// Mitsubishi GX Works2 project: 시퀀스 부분 반복 회로 (카운터)   PLC: Q03UDV

PROGRAM MAIN
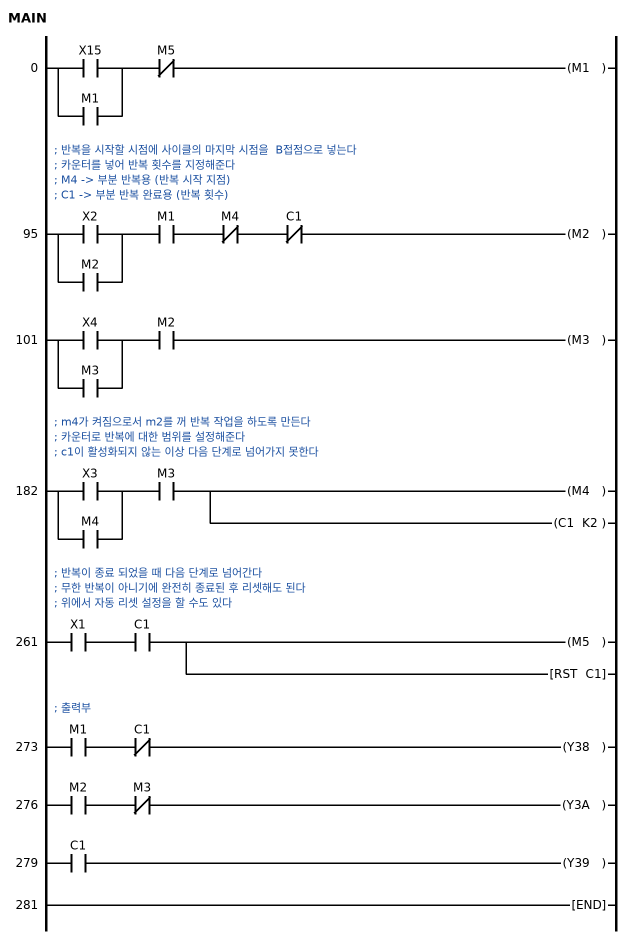
0     LD      X15
      OR      M1
      ANI     M5
      OUT     M1
; 반복을 시작할 시점에 사이클의 마지막 시점을  B접점으로 넣는다
; 카운터를 넣어 반복 횟수를 지정해준다
; M4 -> 부분 반복용 (반복 시작 지점)
; C1 -> 부분 반복 완료용 (반복 횟수)
95    LD      X2
      OR      M2
      AND     M1
      ANI     M4
      ANI     C1
      OUT     M2
101   LD      X4
      OR      M3
      AND     M2
      OUT     M3
; m4가 켜짐으로서 m2를 꺼 반복 작업을 하도록 만든다
; 카운터로 반복에 대한 범위를 설정해준다
; c1이 활성화되지 않는 이상 다음 단계로 넘어가지 못한다
182   LD      X3
      OR      M4
      AND     M3
      OUT     M4
      OUT     C1 K2
; 반복이 종료 되었을 때 다음 단계로 넘어간다
; 무한 반복이 아니기에 완전히 종료된 후 리셋해도 된다
; 위에서 자동 리셋 설정을 할 수도 있다
261   LD      X1
      AND     C1
      OUT     M5
      RST     C1
; 출력부
273   LD      M1
      ANI     C1
      OUT     Y38
276   LD      M2
      ANI     M3
      OUT     Y3A
279   LD      C1
      OUT     Y39
281   END
END_PROGRAM
